INTERFACE I_FunctionCtrl

PROPERTY Busy : BOOL
GET
END_GET
END_PROPERTY

PROPERTY Done : BOOL
GET
END_GET
END_PROPERTY

PROPERTY Error : BOOL
GET
END_GET
END_PROPERTY

PROPERTY ErrorCode : WORD
GET
END_GET
END_PROPERTY

METHOD Execute : BOOL
VAR_INPUT
END_VAR
END_METHOD

PROPERTY Ready : BOOL
GET
END_GET
END_PROPERTY

METHOD Reset : BOOL
VAR_INPUT
END_VAR
END_METHOD

END_INTERFACE

(* stored: Version 1.1.0.1, ProductVersion 3.1.4024.12
   Itf I_FunctionCtrl: Id {75825b88-e051-41e1-bbb8-dba470dbfa85}
   Property Busy: Id {762627fd-1668-4582-b138-af236d08d857}
   Get Get: Id {e83284a1-35e1-49c8-a1d5-a7de831f6808}
   Property Done: Id {b6b16eae-2766-479d-b5a4-225237641aa4}
   Get Get: Id {3747324a-74de-4abd-bb9e-c7ce844f3a91}
   Property Error: Id {ee917f80-b962-4d3b-9b75-bf215e983ec2}
   Get Get: Id {fd7cdf33-ec5b-4539-ad00-a1f8e619c3dd}
   Property ErrorCode: Id {790ee994-ef1f-4260-9e9f-10942df8c7b8}
   Get Get: Id {7adfeff6-cba1-4b46-93f4-6e0e8f7d576b}
   Method Execute: Id {d0740410-8171-4a25-980b-853f7b4191c7}
   Property Ready: Id {f2008cc2-d584-4f85-a508-96e681ebc01b}
   Get Get: Id {93880a20-a6dc-4e63-aa89-8441c74272b3}
   Method Reset: Id {b6773d63-d6c5-4448-8aee-ddd048cc2087} *)
